{attribute 'reflection'}
FUNCTION_BLOCK Tag IMPLEMENTS I_Tag
VAR
	{attribute 'instance-path'} 
    {attribute 'noinit'} 
	_sId			: Strings.Str;
	_nOptionPos		: USINT;
	_nOptionLen		: USINT;
	_nCache			: UDINT;
	_iOwner			: I_TagOwner;
END_VAR

PROPERTY Cache : UDINT
GET
Cache := _nCache;
END_GET
END_PROPERTY

METHOD FB_init : BOOL
VAR_INPUT
	bInitRetains : BOOL; // if TRUE, the retain variables are initialized (warm start / cold start)
	bInCopyCode : BOOL;  // if TRUE, the instance afterwards gets moved into the copy code (online change)
END_VAR
VAR
	i				: INT;
	_sChar			: Strings.Ch;
	
END_VAR
// Delete this name
FOR i := Tc2_Standard.LEN(_sId) TO 1 BY -1 DO
	IF Tc2_Standard.MID(_sId, 1, i) = '.' THEN
		_sId := Tc2_Standard.LEFT(_sId, i - 1);
		EXIT;
	END_IF
END_FOR

// Delete project name
FOR i := 1 TO Tc2_Standard.LEN(_sId) DO
	IF Tc2_Standard.MID(_sId, 1, i) = '.' THEN
		_sId := Tc2_Standard.DELETE(_sId, i, 1);
		EXIT;
	END_IF
END_FOR

// Delete plc name
FOR i := 1 TO Tc2_Standard.LEN(_sId) DO
	IF Tc2_Standard.MID(_sId, 1, i) = '.' THEN
		_sId := Tc2_Standard.DELETE(_sId, i, 1);
		EXIT;
	END_IF
END_FOR

// Replace '[' with '.' and remove ']' 
FOR i := 1 TO Tc2_Standard.LEN(_sId) DO
	_sChar := Tc2_Standard.MID(_sId, 1, i);
	IF _sChar = '[' THEN
		_sId := Tc2_Standard.REPLACE(_sId, '.', 1, i);
	ELSIF _sChar = ']' THEN
		_sId := Tc2_Standard.DELETE(_sId, 1, i);
	END_IF
END_FOR

_sId := Tc2_Utilities.F_ToLCase(_sID);
END_METHOD

METHOD GetId : Strings.Str
VAR_INPUT
END_VAR
IF _nOptionPos <> 0 THEN
	GetId := Tc2_Standard.DELETE(_sId, _nOptionLen + 1, _nOptionPos); 
ELSE
	GetId := _sId;
END_IF
END_METHOD

METHOD Join : Results.Result
VAR_INPUT
	iOwner		: I_TagOwner;
	nCache		: UDINT;
END_VAR
IF iOwner = 0 THEN
	Join := Results.Err.Itf0;
	RETURN;
END_IF

IF _iOwner <> 0 THEN
	Join := Results.Err.ItfEq;
	RETURN;
END_IF

_iOwner := iOwner;
_nCache := nCache;
Join := Results.Ok;
END_METHOD

METHOD Leave : Results.Result
VAR_INPUT
	iOwner		: I_TagOwner;
END_VAR
IF iOwner = 0 THEN
	Leave := Results.Err.Itf0;
	RETURN;
END_IF

IF _iOwner <> iOwner THEN
	Leave := Results.Err.ItfEq;
	RETURN;
END_IF

_iOwner := 0;
Leave := Results.Ok;
END_METHOD

PROPERTY Option : Strings.Str
GET
VAR
	i				: INT;
END_VAR
IF _nOptionPos <> 0 THEN
	Option := Tc2_Standard.DELETE(_sId, _nOptionPos, 1); 
ELSE
	Option := '';
END_IF
END_GET
SET
IF Option <> '' THEN
    _nOptionLen := INT_TO_USINT(Tc2_Standard.LEN(Option));    
    IF _nOptionPos <> 0 THEN
        _sId := Tc2_Standard.LEFT(_sId, _nOptionPos);
        _sId := Tc2_Standard.CONCAT(_sId, Option);
    ELSE
        // The option does not exist, so we append it
        _nOptionPos := INT_TO_USINT(Tc2_Standard.LEN(_sId) + 1);
        _sId := Tc2_Standard.CONCAT(_sId, '.');
        _sId := Tc2_Standard.CONCAT(_sId, Option);
    END_IF
ELSIF _nOptionPos <> 0 THEN
    _sId := Tc2_Standard.LEFT(_sId, _nOptionPos - 1);
    _nOptionPos := 0;
END_IF
END_SET
END_PROPERTY

PROPERTY Owner : I_TagOwner
GET
Owner := _iOwner;
END_GET
END_PROPERTY

PROPERTY Self : I_Tag
GET
Self := THIS^;
END_GET
END_PROPERTY

END_FUNCTION_BLOCK

(* stored: Version 1.1.0.1
   POU Tag: Id {62ca4927-4975-427b-9d4f-c107a36fa9ac}, SpecialFunc None
   Property Cache: Id {31e567c1-84ea-46eb-9fdc-bbaff4cca7d0}
   Get Get: Id {f25a9d69-6d6e-4469-879c-93f392d59d1c}
   Method FB_init: Id {6d8fbfb8-5809-4a8b-b251-034e8e055ab1}
   Method GetId: Id {1e7c2d46-85b3-4961-9ee8-452fbfd30f72}
   Method Join: Id {ec7b1158-e43b-430d-9d25-e55222f877f1}
   Method Leave: Id {7703d5eb-5cdb-4692-bbc5-0b272eb249d2}
   Property Option: Id {a87258c3-8a4d-4f79-bed1-5cd6eb67bb5c}
   Get Get: Id {d70a5443-5cec-419b-a600-5b201698b86d}
   Set Set: Id {711c7481-b132-44f6-9eb4-329138f9c5dc}
   Property Owner: Id {7d22447e-9b37-49ee-8dfa-1abfd149d2a7}
   Get Get: Id {0ff4112d-ce28-467a-ac12-a9c0ee0f1f20}
   Property Self: Id {2bf468fc-144d-481b-af97-9bbf22caa508}
   Get Get: Id {735cc7bd-2863-42f9-8ff2-a104770ddc52} *)
